FUNCTION_BLOCK FB_Robotsteuerung
VAR_INPUT
	bEnable   : BOOL;
  	bExecute  : BOOL;
	bxposition : REAL;
	byposition : REAL;
	bzposition : REAL;
	
	bxEndschalter: BOOL;
	byEndschalter: BOOL;
	bzEndschalter: BOOL;
	bGEndschalter: BOOL;
	
	
END_VAR
VAR_OUTPUT
	estate : eBetriebszustand;
	movedone : BOOL;
END_VAR
VAR
	fbXAchse : FB_Manachse;
	fbYAchse : FB_Manachse;
	fbZAchse : FB_Manachse;
	fbGAchse : FB_ManAchse;  
	nstate : INT := 0;
	currentpos : REAL;
	
	
END_VAR
VAR_IN_OUT
    // Achsen-Referenzen 
    ax_ManX    : AXIS_REF;   
    ax_ManY    : AXIS_REF;   
    ax_ManZ    : AXIS_REF;  
	ax_ManG    : AXIS_REF;   
END_VAR

fbXAchse(
	benable:= , 
	bexecute:= , 
	bEndschalter:= bxEndschalter, 
	rPosition:= bxposition, 
	rVel:= 30, 
	estate=> , 
	ax:= ax_ManX);
	
fbYAchse(
	benable:= , 
	bexecute:= , 
	bEndschalter:= bxEndschalter, 
	rPosition:= byposition, 
	rVel:= 30, 
	estate=> , 
	ax:= ax_ManY);
	
fbZAchse(
	benable:= , 
	bexecute:= , 
	bEndschalter:= bzEndschalter, 
	rPosition:= bzposition, 
	rVel:= 30, 
	estate=> , 
	ax:= ax_ManZ );
	
fbGAchse(
	benable:= , 
	bexecute:= , 
	bEndschalter:= bGEndschalter, 
	rPosition:= , 
	rVel:= 10, 
	estate=> , 
	ax:= ax_ManG);
	
	
CASE nstate OF
	0: //off
	estate := eBetriebszustand.off;
	fbxAchse.benable := FALSE;
	fbyAchse.benable := FALSE;
	fbzAchse.benable := FALSE;
	fbGAchse.benable := FALSE;
	
	IF bEnable THEN
		nstate := 10;
	END_IF
	
	10: //INIT
	fbxAchse.benable := TRUE;
	fbyAchse.benable := TRUE;
	fbzAchse.benable := TRUE;
	fbGAchse.benable := TRUE;
	
	IF fbxAchse.estate = eBetriebszustand.ready AND 
		fbyAchse.estate = eBetriebszustand.ready AND
		fbzAchse.estate = eBetriebszustand.ready THEN
		nstate := 20;
		currentpos := 0.0;
	END_IF
	
	20: // Ready
	eState := eBetriebszustand.ready;
	fbxAchse.benable := TRUE;
	fbyAchse.benable := TRUE;
	fbzAchse.benable := TRUE;
	fbGAchse.benable := TRUE;
	
	IF bexecute AND currentpos < 50.0 THEN
		nstate := 30;
	ELSIF bexecute AND currentpos > 50.0 THEN
		nstate := 60;
	END_IF
	
	30: // MOVEXY
	eState := eBetriebszustand.production;
	fbXAchse.bexecute := TRUE;
	fbYAchse.bexecute := TRUE;
	
	IF fbXAchse.estate = eBetriebszustand.done AND 
		fbYAchse.estate = eBetriebszustand.done THEN
		fbXAchse.bexecute := FALSE;
		fbYAchse.bexecute := FALSE;
		nstate := 40;
	END_IF
	
	40: //MoveZ
	eState := eBetriebszustand.production;
	fbZAchse.bexecute := TRUE;
	
	IF fbZAchse.estate = eBetriebszustand.done THEN
		currentpos := bzposition;
		fbXAchse.bexecute := FALSE;
		nstate  := 50;
	END_IF
	
	50: //Gripper oeffnen
	eState := eBetriebszustand.production;
	fbGAchse.rPosition := 0;
	fbGAchse.bexecute := TRUE;
	
	IF fbGAchse.estate = eBetriebszustand.done THEN
		fbGAchse.bexecute := FALSE;
		nstate := 100;
	END_IF
	
	60: //Gripper oeffnen
	eState := eBetriebszustand.production;
	fbGAchse.rPosition := 8;
	fbGAchse.bexecute := TRUE;
	
	IF fbGAchse.estate = eBetriebszustand.done THEN
		fbGAchse.bexecute := FALSE;
		nstate := 70;
	END_IF	
	
	70: //MoveZ
	eState := eBetriebszustand.production;
	fbZAchse.bexecute := TRUE;
	
	IF fbZAchse.estate = eBetriebszustand.done THEN
		currentpos := bzposition;
		fbXAchse.bexecute := FALSE;
		nstate  := 100;
	END_IF
	
	100: //done
	eState := eBetriebszustand.done;
	
	IF NOT bexecute THEN
		nstate := 20;
	END_IF
	
END_CASE

END_FUNCTION_BLOCK

(* stored: Version 1.1.0.1, ProductVersion 3.1.4024.15
   POU FB_Robotsteuerung: Id {d3df2f2e-da95-4e7a-9ca9-813288b88a86}, SpecialFunc None *)
